# EPICS substitutions: lsredis/iocBoot/iocvxWorks/fb_epid.substitutions
# $Id: fb_epid.substitutions 14505 2012-02-29 21:25:07Z jemian $

file "$(OPTICS)/opticsApp/Db/fb_epid.db"
  {
    {
        P=lsredis:epid1,
	IN=lsredis:epid1:sim.VAL,
	OUT=lsredis:epid1:sim.D,
	MODE=PID,
	CALC=A,
	PERMIT1="lsredis:epid1:on.VAL",
	PERMIT2="",
	PERMIT3="",
	PERMIT4=""
    }
  }
